// Mitsubishi GX Works2 project: FX3U   PLC: FX3U/FX3UC

// global labels: Global1
VAR_GLOBAL
  XXLimitN AT M8344 : BOOL;
  XXLimitP AT M8343 : BOOL;
  XXBusy AT M8340 : BOOL;
  XXInterruptInverse AT M8347 : BOOL;
  XXPos AT D8340 : DINT;
  XXAccelTime AT D8348 : INT;
  XXDecelTime AT D8349 : INT;
  XXPosView AT D0 : DINT;
  XXTarPos AT D2 : DINT;
  XXFeed AT D4 : DINT;
  XXPPR AT D6 : DINT;
  XXTarR AT M0 : BOOL;
  XXTarRSkip AT D8 : INT;
  XXOn AT M1 : BOOL;
  XXRun AT M2 : BOOL;
  XXDirection AT M3 : BOOL;
  XXReady AT M4 : BOOL;
  XXReadyI AT X004 : BOOL;
  XXPulseO AT Y000 : BOOL;
  XXDirectionO AT Y004 : BOOL;
  XXOnO AT Y010 : BOOL;
  YYLimitN AT M8354 : BOOL;
  YYLimitP AT M8353 : BOOL;
  YYBusy AT M8350 : BOOL;
  YYInterruptInverse AT M8357 : BOOL;
  YYPos AT D8350 : DINT;
  YYAccelTime AT D8358 : INT;
  YYDecelTime AT D8359 : INT;
  YYPosView AT D9 : DINT;
  YYTarPos AT D11 : DINT;
  YYFeed AT D13 : DINT;
  YYPPM AT D15 : DINT;
  YYTarR AT M5 : BOOL;
  YYTarRSkip AT D17 : INT;
  YYOn AT M6 : BOOL;
  YYRun AT M7 : BOOL;
  YYDirection AT M8 : BOOL;
  YYReady AT M9 : BOOL;
  YYReadyI AT X005 : BOOL;
  YYPulseO AT Y001 : BOOL;
  YYDirectionO AT Y005 : BOOL;
  YYOnO AT Y011 : BOOL;
  ZZLimitN AT M8364 : BOOL;
  ZZLimitP AT M8363 : BOOL;
  ZZBusy AT M8360 : BOOL;
  ZZInterruptInverse AT M8367 : BOOL;
  ZZPos AT D8360 : DINT;
  ZZAccelTime AT D8368 : INT;
  ZZDecelTime AT D8369 : INT;
  ZZPosView AT D18 : DINT;
  ZZTarPos AT D20 : DINT;
  ZZFeed AT D22 : DINT;
  ZZPPR AT D24 : DINT;
  ZZTarR AT M10 : BOOL;
  ZZTarRSkip AT D26 : INT;
  ZZOn AT M11 : BOOL;
  ZZRun AT M12 : BOOL;
  ZZDirection AT M13 : BOOL;
  ZZReady AT M14 : BOOL;
  ZZReadyI AT X006 : BOOL;
  ZZPulseO AT Y002 : BOOL;
  ZZDirectionO AT Y006 : BOOL;
  ZZOnO AT Y012 : BOOL;
  AxisXState AT D27 : INT;
  AxisXStateNext AT M15 : BOOL;
  AxisYState AT D28 : INT;
  AxisYStateNext AT M16 : BOOL;
  AxisZState AT D29 : INT;
  AxisZStateNext AT M17 : BOOL;
  AutoI AT X017 : BOOL;
END_VAR

// task Task_01 (event TRUE, interval 0, priority 31): POU_01

PROGRAM POU_01
SET(M8002 AND AutoI, XXOn);
SET(M8002 AND AutoI, YYOn);
SET(M8002 AND AutoI, ZZOn);
ZRST(M8002, AxisXState, AxisZState);

(*|||||||||||||||*)
INC(AxisXStateNext, AxisXState);
INC(AxisYStateNext, AxisYState);
INC(AxisZStateNext, AxisZState);
ZRST(M8000, AxisXStateNext, AxisZStateNext);
DECO(M8000, AxisXState, 6, M100); DECO(M8000, AxisXState, 6, M1100); ZRST(NOT AutoI OR NOT XXReady, M1100, M1163);
DECO(M8000, AxisYState, 6, M200); DECO(M8000, AxisYState, 6, M1200); ZRST(NOT AutoI OR NOT YYReady, M1200, M1263);
DECO(M8000, AxisZState, 6, M300); DECO(M8000, AxisZState, 6, M1300); ZRST(NOT AutoI OR NOT ZZReady, M1300, M1363);
DECO(M8000, AxisXState, 2, Y20);
DECO(M8000, AxisYState, 2, Y24);
DECO(M8000, AxisZState, 2, Y30);
(*|||||||||||||||*)

(*axis x*)
DMOV(M1100, 20_000, XXTarPos);
DMOV(M1100, 50_000, XXFeed);
SET(M1100, XXRun);
SET(M1100, AxisXStateNext);
(**)
DMOV(M1101, 0, XXTarPos);
DMOV(M1101, 100_000, XXFeed);
SET(M1101, XXRun);
SET(M1101, AxisXStateNext);
(**)
MOV(M1102, 0, AxisXState);
(**)

(*axis y*)
DMOV(M1200, 25_000, YYTarPos);
DMOV(M1200, 50_000, YYFeed);
SET(M1200, YYRun);
SET(M1200, AxisYStateNext);
(**)
DMOV(M1201, 0, YYTarPos);
DMOV(M1201, 100_000, YYFeed);
SET(M1201, YYRun);
SET(M1201, AxisYStateNext);
(**)
MOV(M1202, 0, AxisYState);
(**)

(*axis z*)
DMOV(M1300, 30_000, ZZTarPos);
DMOV(M1300, 50_000, ZZFeed);
SET(M1300, ZZRun);
SET(M1300, AxisZStateNext);
(**)
DMOV(M1301, 0, ZZTarPos);
DMOV(M1301, 100_000, ZZFeed);
SET(M1301, ZZRun);
SET(M1301, AxisZStateNext);
(**)
MOV(M1302, 0, AxisZState);
(**)

(*|||||||||||||||*)
(*XX*)
RST(XXRun AND XXTarPos = XXPos, XXRun);
DDRVA(XXRun, XXTarPos, XXFeed, XXPulseO, XXDirection);
RST(M8029, XXRun);
OUT(XXDirection, XXDirectionO);
INC(NOT XXRun AND NOT XXBusy AND XXTarRSkip < 5, XXTarRSkip);
RST(XXRun, XXTarRSkip);
OUT(XXTarRSkip >= 5, XXTarR);
(*|||||||||||||||*)
(*YY*)
RST(YYRun AND YYTarPos = YYPos, YYRun);
DDRVA(YYRun, YYTarPos, YYFeed, YYPulseO, YYDirection);
RST(M8029, YYRun);
OUT(NOT YYDirection, YYDirectionO);
INC(NOT YYRun AND NOT YYBusy AND YYTarRSkip < 5, YYTarRSkip);
RST(YYRun, YYTarRSkip);
OUT(YYTarRSkip >= 5, YYTarR);
(*|||||||||||||||*)
(*ZZ*)
RST(ZZRun AND ZZTarPos = ZZPos, ZZRun);
DDRVA(ZZRun, ZZTarPos, ZZFeed, ZZPulseO, ZZDirection);
RST(M8029, ZZRun);
OUT(NOT ZZDirection, ZZDirectionO);
INC(NOT ZZRun AND NOT ZZBusy AND ZZTarRSkip < 5, ZZTarRSkip);
RST(ZZRun, ZZTarRSkip);
OUT(ZZTarRSkip >= 5, ZZTarR);
(*|||||||||||||||*)

OUT(XXReadyI AND XXTarR, XXReady);
OUT(YYReadyI AND YYTarR, YYReady);
OUT(ZZReadyI AND ZZTarR, ZZReady);
OUT(XXOn, XXOnO);
OUT(YYOn, YYOnO);
OUT(ZZOn, ZZOnO);
END_PROGRAM
